{attribute clr [RenderIgnore("Manual")]}
TYPE VortexComponent :
STRUCT
	{attribute clr [RenderIgnore("Control", "ShadowControl")]}
	{attribute addProperty Name "<#Vortex bool#>"}
	vortex_bool: BOOL;
	{attribute addProperty Name "<#Vortex wheel#>"}
	{attribute wpf [Container(Layout.Wrap)]}
	vortex_wheel: Wheel;
END_STRUCT
END_TYPE

(* stored: Version 1.1.0.1, ProductVersion 3.1.4024.9
   DUT VortexComponent: Id {d1164489-f28a-4e73-a53f-172456623777} *)
